# EPICS IOC start-up script: soft_iocs/srs/iocBoot/iocdg645/dg645.iocsh
### Stanford Research Systems (SRS) DG645
# You can use the serial port or the network port, as in the main st.cmd.

# Initialize input/output EOS
asynOctetSetInputEos("$(PORT)",0,"\r\n")
asynOctetSetOutputEos("$(PORT)",0,"\n")

# the device actually uses hardware handshaking
asynSetOption($(PORT), 0, "crtscts",   "Y")

## drvAsynDG645(myport,ioport,ioaddr)
#       myport  - Interface asyn port name (i.e. "DG0")
#       ioport  - Comm asyn port name (i.e. "L2")
#       ioaddr  - Comm asyn port addr
#
drvAsynDG645("DG$(R)","$(PORT)",-1);

# Load database
dbLoadRecords("$(DELAYGEN)/db/drvDG645.db","P=$(P),R=$(R),PORT=DG$(R)")
